# EPICS autosave request: ipApp/Db/Keithley2kDMM_mf_channelN_settings.req
#FILE... Keithley2kDMM_mf_channelN_settings.req
#USAGE... Fields for a single channel in Keithley2kDMM_mf.db fields autosave'd.
$(P)$(Dmm)Ch$(Ch)_on_off.VAL
$(P)$(Dmm)ch$(Ch)_mode_sel.VAL
$(P)$(Dmm)Ch$(Ch)_raw.DESC
file "scalcout_settings.req", P=$(P)$(Dmm)Ch$(Ch)_calc
